FUNCTION_BLOCK PUBLIC RestorePreviousAutomaticState
VAR_INPUT
END_VAR
VAR_OUTPUT
END_VAR
VAR
	RotationRestored: BOOL := FALSE;
	LiftingRestored: BOOL := FALSE;
	ExtensionRestored: BOOL := FALSE;
	GripRestored: BOOL := FALSE;
	DelayTimer: TON; // Timer instance
	
	MotorDirectionEnum: MovementDirection;	// for better clarity on the direction 0 and 1
	MovementEnum: Movement;	// for better clarity on the ON/OFF movement of the motors
END_VAR

IF IO.PreviousManualMode THEN
	Automatic.AllRestored := FALSE;
END_IF

// reset:
Restore(RotationRestored, Automatic.RotationPositionAuto, Automatic.RotationPositionCurrent, 
		Automatic.SafetyRON, Automatic.RCurrentlyMoving, IO.MotorRotationDirection, IO.MotorRotation);

Restore(LiftingRestored, Automatic.LiftingPositionAuto, Automatic.LiftingPositionCurrent, 
		Automatic.SafetyLON, Automatic.LCurrentlyMoving, IO.MotorLiftingDirection, IO.MotorLifting);

Restore(ExtensionRestored, Automatic.ExtensionPositionAuto, Automatic.ExtensionPositionCurrent,
		Automatic.SafetyEON, Automatic.ECurrentlyMoving, IO.MotorExtensionDirection, IO.MotorExtension);

Restore(GripRestored, Automatic.GripPositionAuto, Automatic.GripPositionCurrent,
		Automatic.SafetyGON, Automatic.GCurrentlyMoving, IO.MotorGripDirection, IO.MotorGrip);


// if all restored then go on to execute recipes in AutomaticControl:
IF RotationRestored AND LiftingRestored AND ExtensionRestored AND GripRestored THEN
	DelayTimer(IN := TRUE, PT := T#1S); // Start the timer with a n-second delay
	IF DelayTimer.Q THEN
		IO.PreviousManualMode := FALSE;
		Automatic.AllRestored := TRUE;
		
		RotationRestored := FALSE;
		ExtensionRestored := FALSE;
		LiftingRestored := FALSE;
		GripRestored := FALSE;
		Automatic.RCurrentlyMoving := FALSE;
		Automatic.ECurrentlyMoving := FALSE;
		Automatic.LCurrentlyMoving := FALSE;
		Automatic.GCurrentlyMoving := FALSE;
		DelayTimer(IN := FALSE); // Reset the timer
    END_IF
ELSE
    DelayTimer(IN := FALSE); // Ensure the timer is reset if the conditions are not met
END_IF

END_FUNCTION_BLOCK

(* stored: Version 1.1.0.1, ProductVersion 3.1.4024.13
   POU RestorePreviousAutomaticState: Id {bf2e792f-bc3c-4ce2-afd6-05125fa35279}, SpecialFunc None *)
